{attribute addProperty BoxType "EPP6002-0002-0018"}
{attribute addProperty Id "COM_TxPDO_Map_Inputs_ChannelAT %I*ARRAY[0..1] OF COM_TxPDO_Map_Inputs_Channel_18212A5E384480COM_RxPDO_Map_Outputs_ChannelAT %Q*ARRAY[0..1] OF COM_RxPDO_Map_Outputs_Channel_F536B385384480WcStateAT %I*WcState_F855686C1620InfoDataAT %I*InfoData_BC63D37F80100"}
{attribute addProperty CRC "4014037091"}
{attribute addProperty SizeInBites "864"}
{attribute addProperty SizeInBytes "108"}
TYPE EPP6002_E45E7FFD :
STRUCT
	{attribute addProperty Name "COM_TxPDO_Map_Inputs_Channel"}
	COM_TxPDO_Map_Inputs_Channel : ARRAY[0..1] OF COM_TxPDO_Map_Inputs_Channel_18212A5E;
	{attribute addProperty Name "COM_RxPDO_Map_Outputs_Channel"}
	COM_RxPDO_Map_Outputs_Channel : ARRAY[0..1] OF COM_RxPDO_Map_Outputs_Channel_F536B385;
	{attribute addProperty Name "WcState"}
	WcState : WcState_F855686C;
	{attribute addProperty Name "InfoData"}
	InfoData : InfoData_BC63D37F;
END_STRUCT
END_TYPE

(* stored: Version 1.2.0.0, ProductVersion 3.1.4024.9
   DUT EPP6002_E45E7FFD: Id {505d403a-f613-4773-92c8-afa00efde301} *)
